TYPE E_FlapState :
(
    IdleClosed := 0,
    Opening    := 10,
    Opened     := 20,
    Closing    := 30,
    Fault      := 90   // 🔥 nowy stan
);
END_TYPE

(* stored: Version 1.1.0.1, ProductVersion 3.1.4024.16
   DUT E_FlapState: Id {84a26ebd-5ee0-46d3-b9d4-b964732945a6} *)
